FUNCTION_BLOCK FB_FieldCodecFixed64 IMPLEMENTS I_FieldCodec
VAR_INPUT
END_VAR
VAR_OUTPUT
END_VAR
VAR
    nValue : ULINT;
END_VAR

METHOD CalculatePackedDataSize : HRESULT
VAR_INPUT CONSTANT
	anyFirstElem	: T_Any;
	nLength	        : UDINT;        // items to write
END_VAR
VAR_OUTPUT
    nPackedDataSize : UDINT;
END_VAR
VAR
    anyItem         : T_ANY;
    i               : UDINT;
    nValue          : LINT;
END_VAR
anyItem := anyFirstElem;

IF nLength < 1 THEN
    nPackedDataSize := 0;
    RETURN;
END_IF

FOR i := 0  TO nLength - 1 DO
    anyItem.pValue := anyFirstElem.pValue + (i * TO_UDINT(anyFirstElem.diSize)); 
    nValue := PLINT_TO_LINT(anyItem.pValue);
    nPackedDataSize := nPackedDataSize + F_ComputeFixed64Size(TO_ULINT(nValue));
END_FOR
END_METHOD

METHOD IsPackedRepeatedField : BOOL
VAR_INPUT
	nTag	: UDINT;
END_VAR
IsPackedRepeatedField := F_IsPackedRepeatedField(nTag);
END_METHOD


METHOD ValueReader : HRESULT
VAR_INPUT
    stBuffer : ST_Span;
END_VAR
VAR_IN_OUT
	stState	: ST_ParserInternalState;
END_VAR
VAR_OUTPUT
	anyOut	: T_Any;
END_VAR

ValueReader := F_ParseRawLittleEndian64(stBuffer, stState, nValue=> nValue);
anyOut := F_ToAnyType(anyArg:= nValue);
END_METHOD

METHOD ValueWriter : HRESULT
VAR_IN_OUT
	aBuffer	: ARRAY [*] OF BYTE;
END_VAR
VAR_IN_OUT
	stState	: ST_WriterInternalState;
END_VAR
VAR_INPUT
    anyIn : T_ANY;
END_VAR
VAR
    nValue  : LINT;
END_VAR

nValue := PLINT_TO_LINT(anyIn.pValue);
ValueWriter := F_WriteFixed64(aBuffer, stState, TO_ULINT(nValue));
END_METHOD

END_FUNCTION_BLOCK

(* stored: Version 1.1.0.1
   POU FB_FieldCodecFixed64: Id {a0e96d7d-6cca-454c-9525-7d7610089c1f}, SpecialFunc None
   Method CalculatePackedDataSize: Id {da1b4252-ae08-49e8-b7f0-4ce25c46710d}
   Method IsPackedRepeatedField: Id {7e5f79c9-62f6-4994-a350-1b19d8258d4b}
   Method ValueReader: Id {fb5d9211-3c3e-44d6-bdfb-b82f24425a6a}
   Method ValueWriter: Id {e9309791-3d82-4fc3-a2bd-0a2e19850683} *)
